# EPICS autosave request: ADApp/Db/andor3_settings.req
$(P)$(R)FrameRate
$(P)$(R)PreAmpGain
$(P)$(R)ReadoutRate
$(P)$(R)Overlap
$(P)$(R)NoiseFilter
$(P)$(R)PixelEncoding
$(P)$(R)A3Binning
$(P)$(R)A3ShutterMode
$(P)$(R)SensorCooling
$(P)$(R)TempControl
$(P)$(R)FanSpeed
